# EPICS autosave request: softGlueApp/Db/HistScal_settings.req
$(P)$(H)HistScal-$(N)_desc
$(P)$(H)HistScal-$(N)_EN_Signal
$(P)$(H)HistScal-$(N)_SYNC_Signal
$(P)$(H)HistScal-$(N)_CLK_Signal
$(P)$(H)HistScal-$(N)_DET_Signal
$(P)$(H)HistScal-$(N)_CLEAR_Signal
#$(P)$(H)HistScal-$(N)_READ_Signal
$(P)$(H)HistScal-$(N)_DET2_Signal
#$(P)$(H)HistScal-$(N)_MODE_Signal
